TYPE U_OdriveSetAxisStateBytes :
UNION
    stSetAxisState : ST_OdriveSetAxisState;
    aBytes : ARRAY[0..3] OF BYTE;
END_UNION
END_TYPE

(* stored: Version 1.1.0.1
   DUT U_OdriveSetAxisStateBytes: Id {af17718a-55d7-45a5-8856-cfe3cfcc3c14} *)
